(* Schneider Machine Expert - Basic project Timer 2, file version 1.7.0.0 *)
(* ProjectInformations: Name=New project *)

HARDWARE
  Cpu 0: TM221M32TK
  EthernetConfiguration: NetworkName=M221, IpAllocationMode=FixedAddress, IpAddress=0.0.0.0, SubnetMask=0.0.0.0
  SerialLineConfiguration: Baud=Baud19200, Parity=ParityEven, DataBits=DataBits8, StopBits=StopBits1, PhysicalMedium=PhysicalMediumRs485, TransmissionMode=TransmissionModeModbusRtu, SlaveId=1, Addressing=SlaveAddressing
  MastTask: UsePeriodScanMode=false, PeriodScan=100
  FastTask: Period=255
  CpuBehavior: StartingMode=StartAsPreviousState, AutoSaveRamOnEeprom=true, WatchdogPeriod=250

SYMBOLS  (address, symbol, comment, settings)
  %TM0        "T1"  [Preset=10]
  %TM1        "T2"  [Preset=10]
  %TM2        "t3"  [Preset=15]
  %TM3        "t4"  [Preset=5]
  %I0.0       "Auto"
  %I0.1       "Manual"
  %I0.2       "S1"
  %I0.3       "S2"
  %Q0.0       "P03A"
  %Q0.1       "P03B"
  %IW0.0      [Type=Type_0_10V, Scope=Scope_Normal, Minimum=0, Maximum=1000]
  %IW0.1      [Type=Type_0_10V, Scope=Scope_Normal, Minimum=0, Maximum=1000]

POU New POU
  (* SectionNumber=1 *)

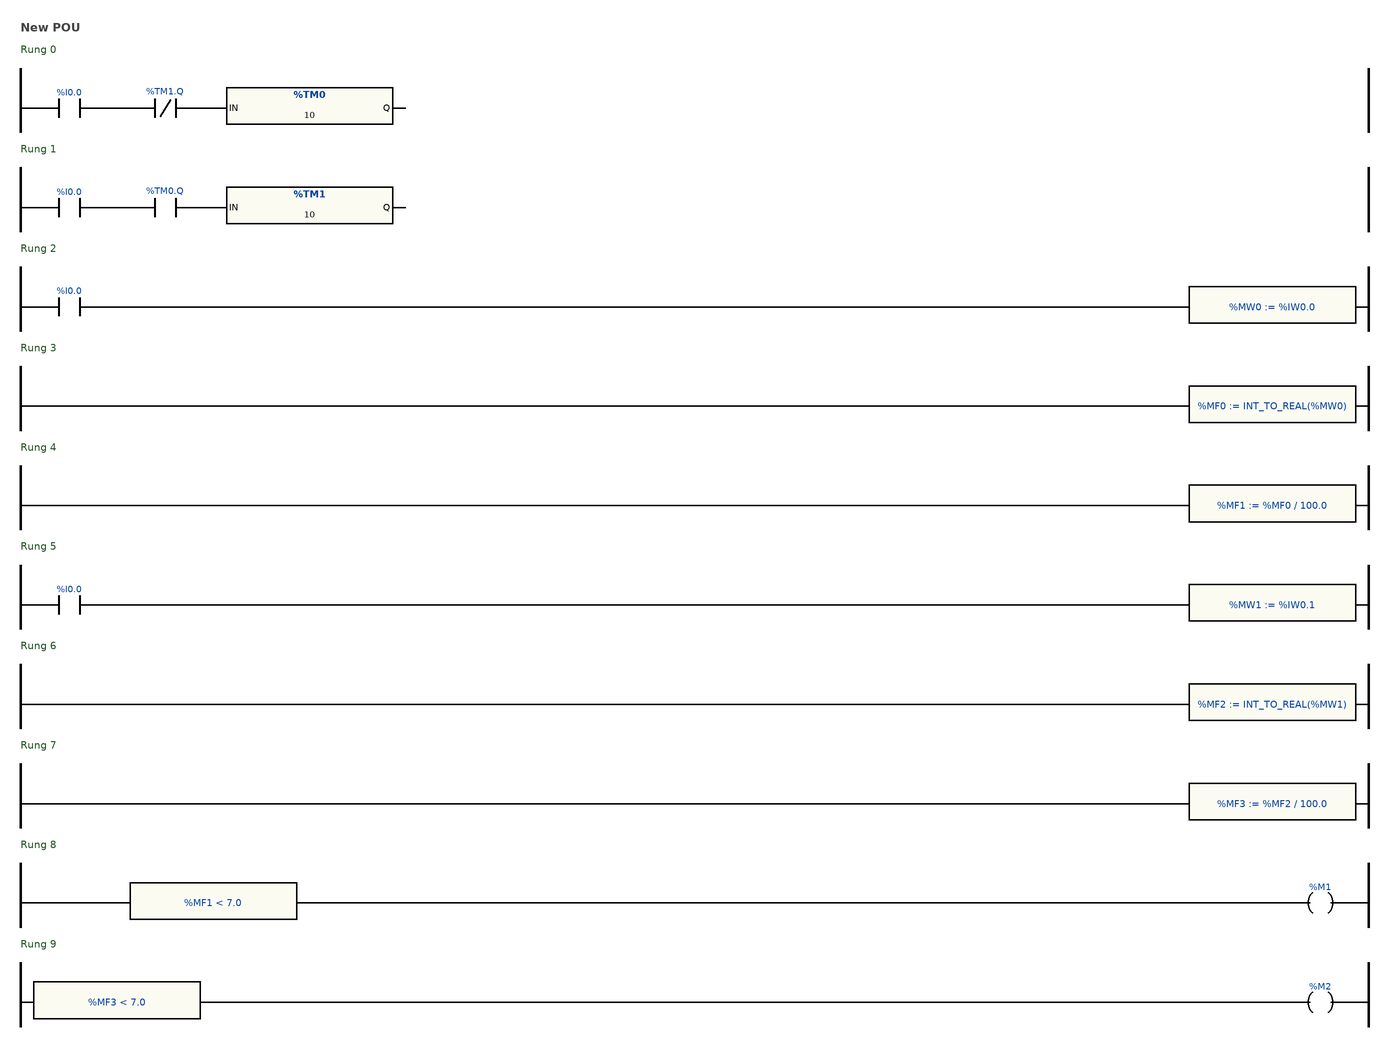

// Rung 0
  BLK %TM0
  LD %I0.0
  ANDN %TM1.Q
  IN
  END_BLK
  // as ST:
  //   %TM0(IN := %I0.0 AND NOT %TM1.Q);

// Rung 1
  BLK %TM1
  LD %I0.0
  AND %TM0.Q
  IN
  END_BLK
  // as ST:
  //   %TM1(IN := %I0.0 AND %TM0.Q);

// Rung 2
  LD %I0.0
  [ %MW0 := %IW0.0 ]
  // as ST:
  //   IF %I0.0 THEN %MW0 := %IW0.0; END_IF;

// Rung 3
  LD 1
  [ %MF0 := INT_TO_REAL ( %MW0 ) ]
  // as ST:
  //   %MF0 := INT_TO_REAL ( %MW0 );

// Rung 4
  LD 1
  [ %MF1 := %MF0 / 100.0 ]
  // as ST:
  //   %MF1 := %MF0  /  100.0;

// Rung 5
  LD %I0.0
  [ %MW1 := %IW0.1 ]
  // as ST:
  //   IF %I0.0 THEN %MW1 := %IW0.1; END_IF;

// Rung 6
  LD 1
  [ %MF2 := INT_TO_REAL ( %MW1 ) ]
  // as ST:
  //   %MF2 := INT_TO_REAL ( %MW1 );

// Rung 7
  LD 1
  [ %MF3 := %MF2 / 100.0 ]
  // as ST:
  //   %MF3 := %MF2  /  100.0;

// Rung 8
  LD [ %MF1 < 7.0 ]
  ST %M1
  // as ST:
  //   %M1 := %MF1 < 7.0;

// Rung 9
  LD [ %MF3 < 7.0 ]
  ST %M2
  // as ST:
  //   %M2 := %MF3 < 7.0;

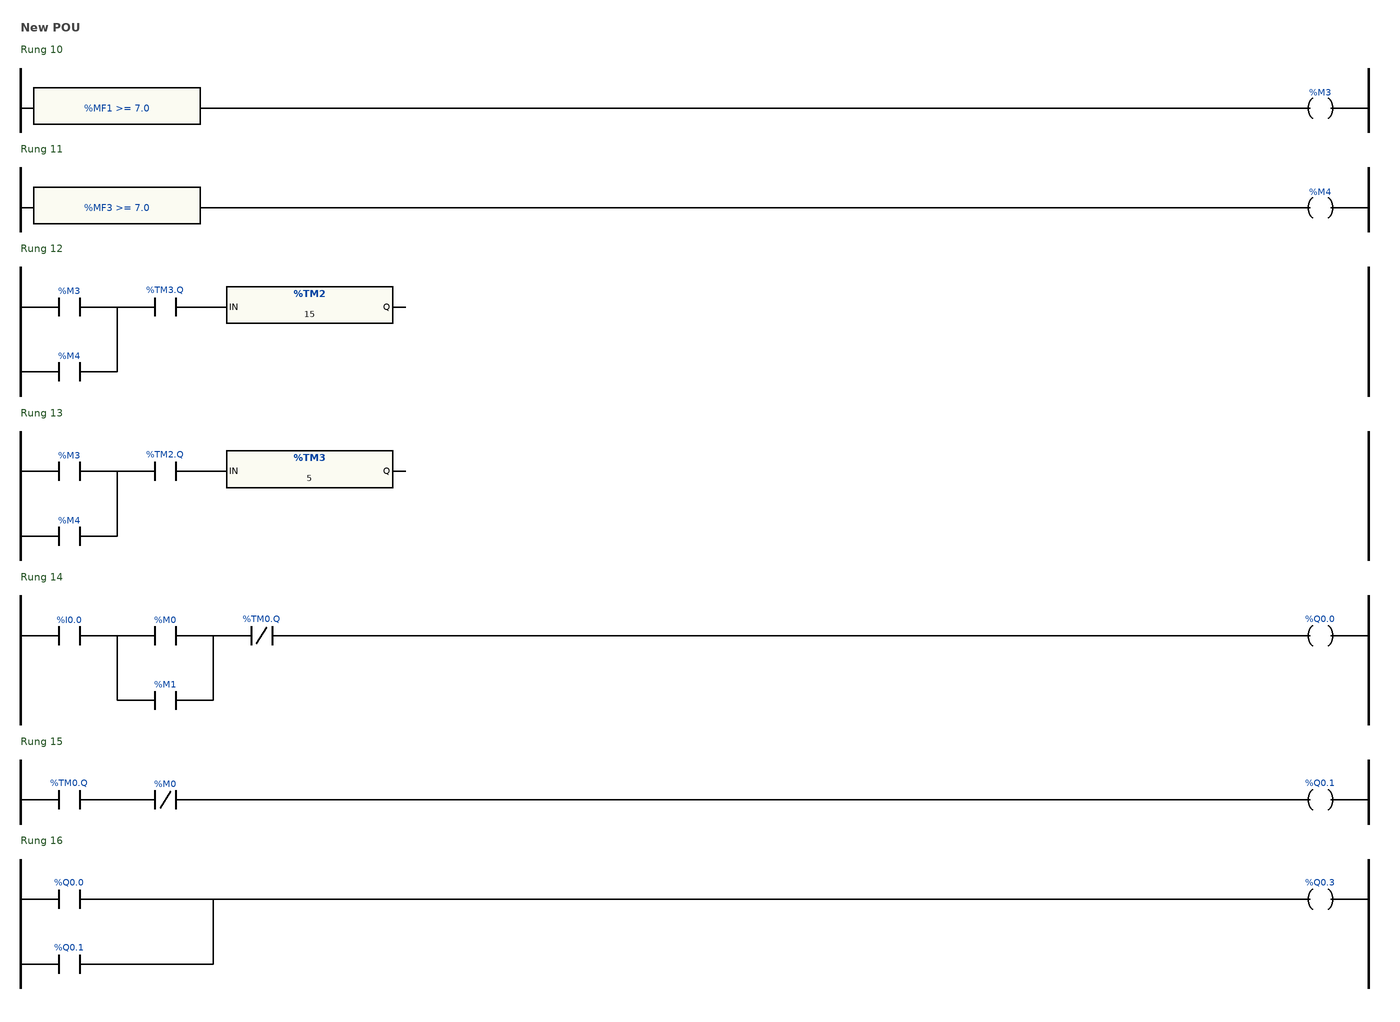

// Rung 10
  LD [ %MF1 >= 7.0 ]
  ST %M3
  // as ST:
  //   %M3 := %MF1 >= 7.0;

// Rung 11
  LD [ %MF3 >= 7.0 ]
  ST %M4
  // as ST:
  //   %M4 := %MF3 >= 7.0;

// Rung 12
  BLK %TM2
  LD %M3
  OR %M4
  AND %TM3.Q
  IN
  END_BLK
  // as ST:
  //   %TM2(IN := (%M3 OR %M4) AND %TM3.Q);

// Rung 13
  BLK %TM3
  LD %M3
  OR %M4
  AND %TM2.Q
  IN
  END_BLK
  // as ST:
  //   %TM3(IN := (%M3 OR %M4) AND %TM2.Q);

// Rung 14
  LD %I0.0
  AND( %M0
  OR %M1
  )
  ANDN %TM0.Q
  ST %Q0.0
  // as ST:
  //   %Q0.0 := %I0.0 AND (%M0 OR %M1) AND NOT %TM0.Q;

// Rung 15
  LD %TM0.Q
  ANDN %M0
  ST %Q0.1
  // as ST:
  //   %Q0.1 := %TM0.Q AND NOT %M0;

// Rung 16
  LD %Q0.0
  OR %Q0.1
  ST %Q0.3
  // as ST:
  //   %Q0.3 := %Q0.0 OR %Q0.1;

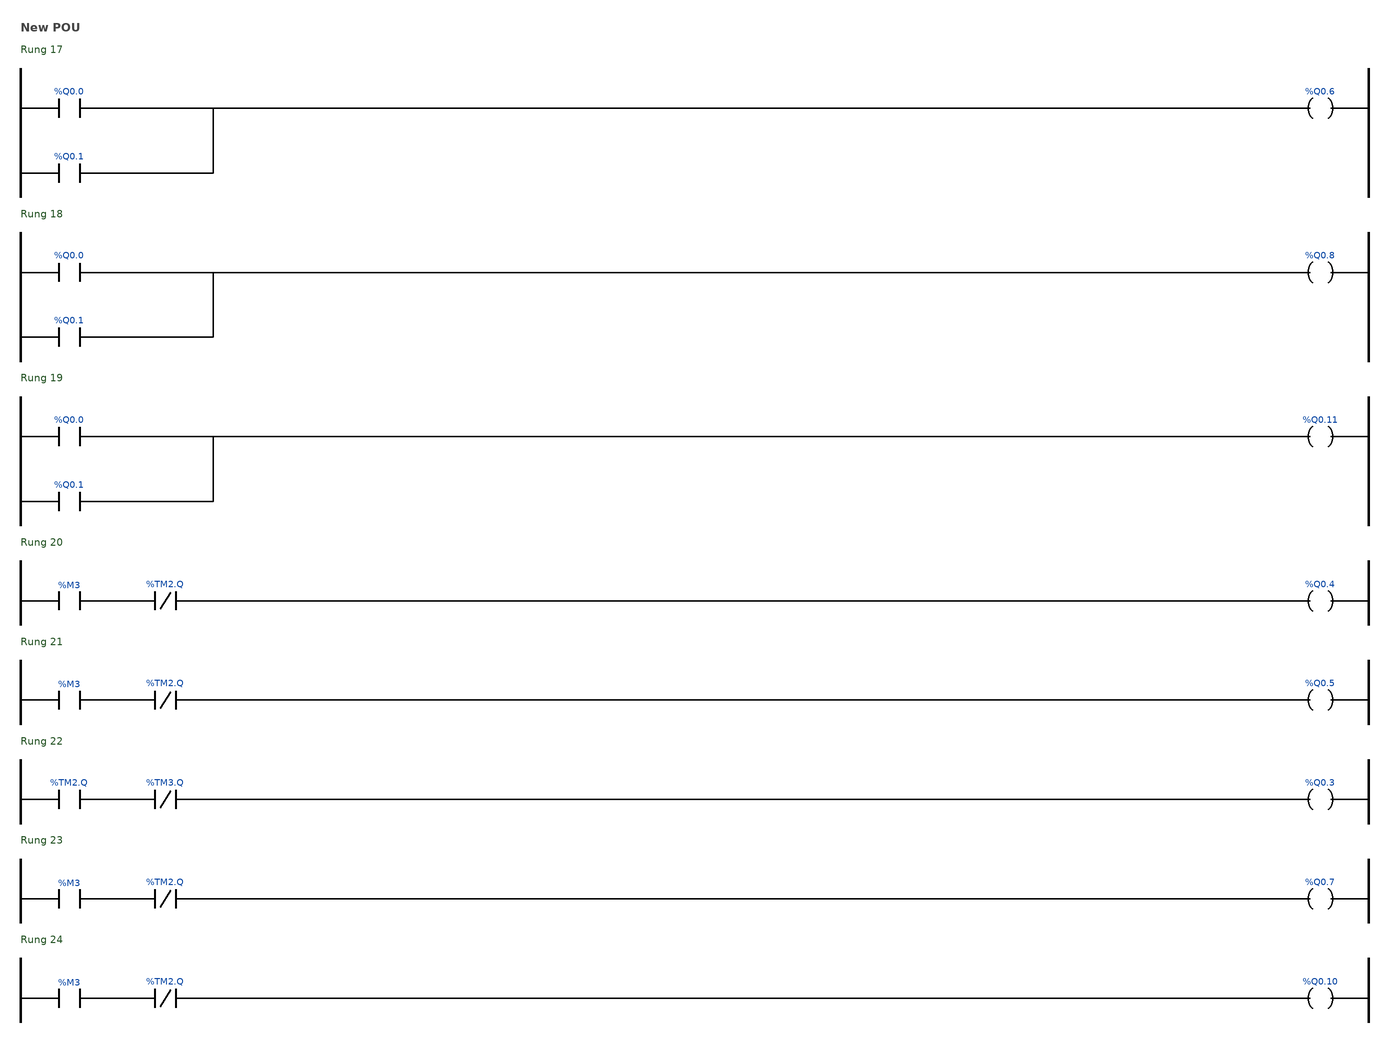

// Rung 17
  LD %Q0.0
  OR %Q0.1
  ST %Q0.6
  // as ST:
  //   %Q0.6 := %Q0.0 OR %Q0.1;

// Rung 18
  LD %Q0.0
  OR %Q0.1
  ST %Q0.8
  // as ST:
  //   %Q0.8 := %Q0.0 OR %Q0.1;

// Rung 19
  LD %Q0.0
  OR %Q0.1
  ST %Q0.11
  // as ST:
  //   %Q0.11 := %Q0.0 OR %Q0.1;

// Rung 20
  LD %M3
  ANDN %TM2.Q
  ST %Q0.4
  // as ST:
  //   %Q0.4 := %M3 AND NOT %TM2.Q;

// Rung 21
  LD %M3
  ANDN %TM2.Q
  ST %Q0.5
  // as ST:
  //   %Q0.5 := %M3 AND NOT %TM2.Q;

// Rung 22
  LD %TM2.Q
  ANDN %TM3.Q
  ST %Q0.3
  // as ST:
  //   %Q0.3 := %TM2.Q AND NOT %TM3.Q;

// Rung 23
  LD %M3
  ANDN %TM2.Q
  ST %Q0.7
  // as ST:
  //   %Q0.7 := %M3 AND NOT %TM2.Q;

// Rung 24
  LD %M3
  ANDN %TM2.Q
  ST %Q0.10
  // as ST:
  //   %Q0.10 := %M3 AND NOT %TM2.Q;

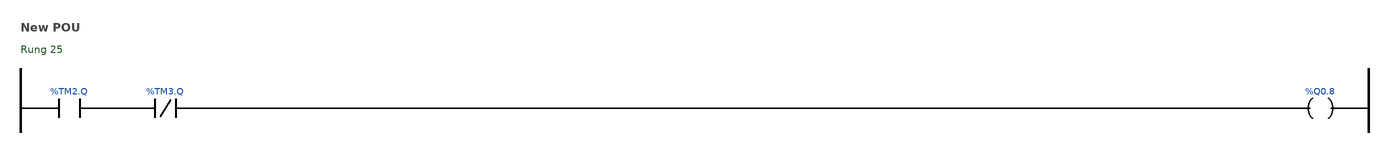

// Rung 25
  LD %TM2.Q
  ANDN %TM3.Q
  ST %Q0.8
  // as ST:
  //   %Q0.8 := %TM2.Q AND NOT %TM3.Q;
